// =============================================================================
// FB_PPC_Controller  —  Plant Power Controller, main block
// -----------------------------------------------------------------------------
// PURPOSE:
//   Orchestrates the entire PPC control loop. Called from OB30 (cyclic interrupt,
//   default 100 ms). Calls six FCs in a fixed order; each FC feeds the next.
//
// CALL ORDER AND DATA FLOW:
//   ①  FC_PPC_InverterMonitor    →  N_Online, PmaxPlant, QmaxPlant
//   ②  FC_PPC_ModeManager        →  Plant_Mode  (LOCAL / REMOTE_IEC / FALLBACK)
//   ③  FC_PPC_RampControl        →  Ramps_Pcmd  (rate-limited P command in kW)
//   ④  FC_PPC_PowerDistribution  →  WSpt, WMode per inverter
//   ⑤  FC_PPC_ReactiveControl    →  Ramps_Qcmd, VArSpt / PFSpt / VArMode per inverter
//   ⑥  FC_PPC_FaultHandler       →  OperMode overrides; AnyFault, AnyDerating, FaultMask
//
// DB39 FIELDS REQUIRED (user must add if not present):
//   Q_RampUp     : REAL    — Q ramp rate up in kVAr/s
//   Q_RampDown   : REAL    — Q ramp rate down in kVAr/s
//   Ramps_Qcmd   : REAL    — mirrored ramped Q command for HMI trending
//   AnyDerating  : BOOL    — mirrored derating alarm flag
//   FaultMask    : WORD    — mirrored per-inverter fault bitmap (bit i = inverter i)
//
// LOCAL MODE:
//   When Plant_Mode = 0 (LOCAL), the OB30 caller is responsible for supplying
//   Cmd_P and Cmd_Q from the HMI DB rather than from the SCADA comms thread.
//   The PLC logic itself does not switch the setpoint source.
//
// FALLBACK RECOVERY (S4 fix):
//   When Plant_Mode transitions from FALLBACK (2) to REMOTE_IEC (1), both
//   Ramps_Pcmd and Ramps_Qcmd are forced to 0. This ensures a clean ramp-up
//   from zero regardless of whether any inverters stayed online during FALLBACK.
//
// CALLED FROM: OB30 (cyclic, 100 ms)
// INSTANCE DB:  assign one DB when placing the FB call in OB30
// =============================================================================

FUNCTION_BLOCK "FB_PPC_Controller"
{ S7_Optimized_Access := 'TRUE' }
VERSION : 0.1

// ─────────────────────────────────────────────────────────────────────────────
// INPUTS  (set by the OB30 network that calls this FB)
// ─────────────────────────────────────────────────────────────────────────────
VAR_INPUT
    // Master enable. FALSE → all inverters commanded to Stop immediately.
    EN_PPC : BOOL;

    // Heartbeat bit from the upstream Modbus/IEC comms thread.
    // Must toggle (0→1 edge) at least once per Watchdog_Timeout period.
    IEC_Watchdog : BOOL;

    // OB30 cycle time in seconds. Default: 0.1 (100 ms).
    CycleTime_s : REAL;

    // Active power target from upstream SCADA / grid operator, in kW.
    // In LOCAL mode: supplied by OB30 caller from HMI DB.
    Cmd_P : REAL;

    // Reactive power target in kVAr. Used when Cmd_VArMode = 1.
    // In LOCAL mode: supplied by OB30 caller from HMI DB.
    Cmd_Q : REAL;

    // Power factor target (e.g. 0.95, 1.00). Used when Cmd_VArMode = 2.
    Cmd_PF : REAL;

    // Reactive control mode: 0 = Off, 1 = Q setpoint, 2 = PF setpoint.
    Cmd_VArMode : INT;

    // TRUE when HMI LOCAL/REMOTE selector is in LOCAL.
    LocalMode_Req : BOOL;
END_VAR

// ─────────────────────────────────────────────────────────────────────────────
// OUTPUTS
// ─────────────────────────────────────────────────────────────────────────────
VAR_OUTPUT
    // TRUE when Plant_Mode = 1 (REMOTE_IEC) — controller active.
    PPC_Active : BOOL;

    // TRUE when any inverter has an active fault, comms error, or PwrOffReas ≠ 0.
    PPC_Fault : BOOL;

    // TRUE when any healthy inverter reports a non-zero derating state.
    AnyDerating : BOOL;

    // Current Plant_Mode (0/1/2). For HMI display.
    Mode_Out : INT;
END_VAR

// ─────────────────────────────────────────────────────────────────────────────
// STATIC  (retained between OB30 cycles)
// ─────────────────────────────────────────────────────────────────────────────
VAR
    Watchdog_TON     : TON;
    Watchdog_LastBit : BOOL;
    Watchdog_Timeout : TIME := T#30S;

    Plant_Mode  : INT;
    Ramps_Pcmd  : REAL;
    Ramps_Qcmd  : REAL;

    // Previous Plant_Mode — used to detect FALLBACK→REMOTE_IEC transition (S4).
    PrevMode : INT;

    // Previous Error state per inverter — for ErrClr one-shot edge detection (S3.3).
    PrevError_Arr : Array[0..9] of BOOL;

    // Previous Enabled state per inverter — for ErrClr re-send on re-enable (M6).
    PrevEnabled_Arr : Array[0..9] of BOOL;
END_VAR

// ─────────────────────────────────────────────────────────────────────────────
// TEMP  (recalculated each OB30 cycle)
// ─────────────────────────────────────────────────────────────────────────────
VAR_TEMP
    WD_EdgeDetected : BOOL;
    WD_Expired      : BOOL;
    N_Online        : INT;
    PmaxPlant       : REAL;
    QmaxPlant       : REAL;
    AnyFault_Tmp    : BOOL;
    FaultMask       : WORD;
END_VAR


BEGIN

    // =========================================================================
    // GUARD: PPC disabled (EN_PPC = FALSE)
    // =========================================================================
    IF NOT #EN_PPC THEN
        "FC_PPC_FaultHandler"(
            Plant_Mode  := #Plant_Mode,
            ForceStop   := TRUE,
            Inverters   := "PPC_Controller".Inverters.PPC_Inverters,
            Ramps_Pcmd  := #Ramps_Pcmd,
            Ramps_Qcmd  := #Ramps_Qcmd,
            PrevError   := #PrevError_Arr,
            PrevEnabled := #PrevEnabled_Arr,
            AnyFault    => #AnyFault_Tmp,
            AnyDerating => #AnyDerating,
            FaultMask   => #FaultMask
        );
        #Plant_Mode := 0;
        #Ramps_Pcmd := 0.0;
        #Ramps_Qcmd := 0.0;
        #PrevMode   := 0;
        // Write outputs
        #PPC_Active  := FALSE;
        #PPC_Fault   := #AnyFault_Tmp;
        #Mode_Out    := 0;
        // Mirror to DB
        "PPC_Controller".Plant_Mode   := 0;
        "PPC_Controller".Ramps_Pcmd   := 0.0;
        "PPC_Controller".Ramps_Qcmd   := 0.0;
        "PPC_Controller".AnyFault     := #AnyFault_Tmp;
        "PPC_Controller".AnyDerating  := #AnyDerating;
        "PPC_Controller".FaultMask    := #FaultMask;
        RETURN;
    END_IF;


    // =========================================================================
    // WATCHDOG — Rising-edge detection and TON timer management
    // =========================================================================
    #WD_EdgeDetected  := #IEC_Watchdog AND NOT #Watchdog_LastBit;
    #Watchdog_LastBit := #IEC_Watchdog;

    IF #WD_EdgeDetected THEN
        #Watchdog_TON(IN := FALSE, PT := #Watchdog_Timeout);
    ELSE
        #Watchdog_TON(IN := TRUE,  PT := #Watchdog_Timeout);
    END_IF;

    #WD_Expired := #Watchdog_TON.Q;


    // =========================================================================
    // ①  FC_PPC_InverterMonitor
    // =========================================================================
    "FC_PPC_InverterMonitor"(
        WRtg_kW   := "PPC_Controller".WRtg_kW,
        Inverters  := "PPC_Controller".Inverters.PPC_Inverters,
        N_Online   => #N_Online,
        PmaxPlant  => #PmaxPlant,
        QmaxPlant  => #QmaxPlant
    );
    "PPC_Controller".Plant_N_Online   := #N_Online;
    "PPC_Controller".Limits_PmaxPlant := #PmaxPlant;
    "PPC_Controller".Limits_QmaxPlant := #QmaxPlant;


    // =========================================================================
    // ②  FC_PPC_ModeManager
    // =========================================================================
    "FC_PPC_ModeManager"(
        WD_Expired    := #WD_Expired,
        LocalMode_Req := #LocalMode_Req,
        Plant_Mode    := #Plant_Mode
    );
    "PPC_Controller".Plant_Mode := #Plant_Mode;

    // ── S4: Reset ramps on FALLBACK → REMOTE_IEC transition ──────────────────
    // Force both ramps to 0 whenever comms recover from FALLBACK, ensuring
    // a clean ramp-up from zero regardless of inverter state during FALLBACK.
    IF (#PrevMode = 2) AND (#Plant_Mode <> 2) THEN
        #Ramps_Pcmd := 0.0;
        #Ramps_Qcmd := 0.0;
    END_IF;
    #PrevMode := #Plant_Mode;


    // =========================================================================
    // ③  FC_PPC_RampControl
    // =========================================================================
    "FC_PPC_RampControl"(
        Targets_P   := #Cmd_P,
        PmaxPlant   := #PmaxPlant,
        P_RampUp    := "PPC_Controller".P_RampUp,
        P_RampDown  := "PPC_Controller".P_RampDown,
        CycleTime_s := #CycleTime_s,
        Plant_Mode  := #Plant_Mode,
        Ramps_Pcmd  := #Ramps_Pcmd
    );
    "PPC_Controller".Ramps_Pcmd := #Ramps_Pcmd;


    // =========================================================================
    // ④  FC_PPC_PowerDistribution
    // =========================================================================
    "FC_PPC_PowerDistribution"(
        Ramps_Pcmd := #Ramps_Pcmd,
        Plant_Mode := #Plant_Mode,
        WRtg_kW    := "PPC_Controller".WRtg_kW,
        Inverters  := "PPC_Controller".Inverters.PPC_Inverters
    );


    // =========================================================================
    // ⑤  FC_PPC_ReactiveControl
    // =========================================================================
    "FC_PPC_ReactiveControl"(
        Plant_VArMode := #Cmd_VArMode,
        Targets_Q     := #Cmd_Q,
        Targets_PF    := #Cmd_PF,
        Plant_Mode    := #Plant_Mode,
        Q_RampUp      := "PPC_Controller".Q_RampUp,
        Q_RampDown    := "PPC_Controller".Q_RampDown,
        CycleTime_s   := #CycleTime_s,
        QmaxPlant     := #QmaxPlant,
        Inverters     := "PPC_Controller".Inverters.PPC_Inverters,
        Ramps_Qcmd    := #Ramps_Qcmd
    );
    "PPC_Controller".Ramps_Qcmd := #Ramps_Qcmd;


    // =========================================================================
    // ⑥  FC_PPC_FaultHandler  (always last)
    // =========================================================================
    "FC_PPC_FaultHandler"(
        Plant_Mode  := #Plant_Mode,
        ForceStop   := FALSE,
        Inverters   := "PPC_Controller".Inverters.PPC_Inverters,
        Ramps_Pcmd  := #Ramps_Pcmd,
        Ramps_Qcmd  := #Ramps_Qcmd,
        PrevError   := #PrevError_Arr,
        PrevEnabled := #PrevEnabled_Arr,
        AnyFault    => #AnyFault_Tmp,
        AnyDerating => #AnyDerating,
        FaultMask   => #FaultMask
    );
    "PPC_Controller".AnyFault    := #AnyFault_Tmp;
    "PPC_Controller".AnyDerating := #AnyDerating;
    "PPC_Controller".FaultMask   := #FaultMask;


    // =========================================================================
    // OUTPUT ASSIGNMENTS
    // =========================================================================
    #Mode_Out   := #Plant_Mode;
    #PPC_Active := (#Plant_Mode = 1);
    #PPC_Fault  := #AnyFault_Tmp;

END_FUNCTION_BLOCK
